{attribute 'GeneratedUsingTerminal: EK1100-0000-0018'}
{attribute addProperty BoxType "EK1100-0000-0018"}
{attribute addProperty Id "Beckhoff_EK18xxEK1122Beckhoff_EK18xxEK1122_F7FACD4D179"}
{attribute addProperty CRC "2297243435"}
{attribute addProperty Size "179"}
TYPE Beckhoff_EK18xx_88ED272B EXTENDS EK1100_1FC0878B :
STRUCT
	{attribute addProperty Name "Beckhoff_EK18xxEK1122"}
	{attribute addProperty PreviousPort "Beckhoff EK18xx : B"}
	Beckhoff_EK18xxEK1122 : Beckhoff_EK18xxEK1122_F7FACD4D;
END_STRUCT
END_TYPE

(* stored: Version 1.2.0.0, ProductVersion 3.1.4024.9
   DUT Beckhoff_EK18xx_88ED272B: Id {59c6ed68-4bef-457b-8fef-bc66b90b7415} *)
